(* CoDeSys 2.3.9.48 project: Dev_Test.pro *)
(* Libraries: Standard.lib 20.5.14 08:13:26, Iecsfc.lib 30.1.13 13:05:12, SYSLIBCALLBACK.LIB 30.1.13 13:05:12, WagoLibModbus_IP_01.lib 12.2.16 11:20:24, SysLibSockets.lib 22.5.14 16:16:32, Wago_MBCFG_ETHERNET_01.lib 1.4.15 14:24:28, Wago_MBCFG_COMMON_01.lib 1.4.15 14:24:28 *)

(* PLC configuration (modules and I/O channels)
AT %IX0.0 [BOOLOnX_I] Ch_1 Digital input
AT %IX0.1 [BOOLOnX_I] Ch_2 Digital input
AT %QX4.0 [BOOLOnX_Q] Ch_1 Digital output
AT %QX4.1 [BOOLOnX_Q] Ch_2 Digital output
AT %QW0 [WORDOnW_Q] Ch_1 Analog output
AT %QW1 [WORDOnW_Q] Ch_2 Analog output
AT %QW2 [WORDOnW_Q] Ch_1 Analog output
AT %QW3 [WORDOnW_Q] Ch_2 Analog output
Modbus variables [PFC200MODBUS] node 1, in %IB0 out %QB0 {PlcStopBehaviour = 1; FiledbusErrorBehaviour = 1; TcpOperation = 1; TcpPort = 502; TcpTimeout = 600; UdpOperation = 1; UdpPort = 502; RtuOperation = 0; NodeId = 1; ResponseTimeout = 5000; Interface = 0; Baud = 115200; StopBits = 1; Parity = 1; FlowCtrl = 0; PhysInterface = 0}
Modbus-Master [MB_MASTER] node 2, in %IB0 out %QB0
*)

(* Task configuration *)
TASK NewTask (PRIORITY := 31, INTERVAL := T#1000ms);
	Test();
	SynchronizerModbusStateHandler_PRG();
	SynchroniserSwitch();
	BUS_status_updater();
	MBCFG_ModbusSlave(
	Voltage_LN=> , 
	Power_L=> , 
	MBCFG_IpAddress=> , 
	MBCFG_Port=> , 
	MBCFG_UnitID=> , 
	MBCFG_TimeOut=> , 
	MBCFG_RequestDelay=> , 
	MBCFG_Error=> , 
	MBCFG_LastJob=> );
END_TASK

(* Global variable list: Global_Variables *)
VAR_GLOBAL

	r_modbus_Synchroniser_state								:	REAL:= 1; (* 0 = deny, 1 = allow, 2 = close request*)
	r_modbus_Synchroniser_Denied_Request					:	BOOL;
	r_modbus_Synchroniser_Close_Request					:	BOOL;

	r_DI_Synchroniser_Close_Request				AT %IX0.0	:	BOOL;
	r_DI_Synchroniser_Denied_Request			AT %IX0.1	:	BOOL;

	r_Synchroniser_Close_Request_Relais		AT %QX0.0:	BOOL;
	r_Synchroniser_Close_Denied_Relais			AT %QX0.1:	BOOL; (* only inplemented if hardware output is available *)

(* Offgridbus frequency to analog Out variables*)
     	r_Battery_Bus_Frequency						:	 REAL;
     	x													:	 REAL:=1;
	r_CHP_Power_Control  							: 	REAL;

(* Mixer en CHP frequency variables*)

	Mixer_0_10V_Analog_Control 							AT %QW0		: REAL;
	EV_Charge_0_10V_Analog_Control 					AT %QW1		: REAL;
	CHP_0_20mA_Analog_Control							AT %QW2 		: REAL;


(*Global variables *)
	arSystemState		AT %MW0			:	ARRAY[1.. 2] OF REAL; 			(* Array containing all the system parameters. Values are accessable through modbus tcp starting from register 12288. REAL uses two registers per variable *)



END_VAR

(* POU SWITCHING RELAIS/Test, ST *)
PROGRAM Test
VAR

	Test :fbSwitchRelaysOnOffGrid;
	a: REAL;
	x: REAL;
END_VAR
x := x+1;
arSystemState[1]  := x;

Test(
	r_Off_Grid_Bus_Frequency:= a ,
	r_Off_Grid_Bus_Voltage:= 250,
	r_On_Grid_Start_Frequency:= 49,
	r_On_Grid_Start_Delay_Time:= 2000,
	r_On_Grid_Minimal_On_Time:= 2000 ,
	r_Off_Grid_Start_Frequency:= 51,
	r_Off_Grid_Start_Delay_Time:= 2000,
	r_Switch_Gap_Time:= 2000,
	r_Off_Grid_Minimal_On_Time:= 2000);
END_PROGRAM

(* POU SWITCHING RELAIS/fbSwitchRelaysOnOffGrid, SFC *)
FUNCTION_BLOCK fbSwitchRelaysOnOffGrid
VAR_INPUT

	r_Off_Grid_Bus_Frequency						:	REAL;
	r_Off_Grid_Bus_Voltage							:	REAL;
	r_On_Grid_Start_Frequency						:	REAL;
	r_On_Grid_Start_Delay_Time					:	REAL;
	r_On_Grid_Minimal_On_Time					:	REAL;
	r_Off_Grid_Start_Frequency						:	REAL;
	r_Off_Grid_Start_Delay_Time					:	REAL;
	r_Switch_Gap_Time								: 	REAL;		(* Time between on and off grid relay switching (dead bus gap) *)
	r_Off_Grid_Minimal_On_Time					:	REAL;

END_VAR
VAR_OUTPUT

	r_On_Grid_Relay									:	BOOL;
	r_Off_Grid_Relay									:	BOOL;

END_VAR
VAR

	r_Checked_On_Grid_Start_Frequency			:	REAL;
	r_Checked_Off_Grid_Start_Frequency			:	REAL;

	t_On_Grid_Start_Delay_Timer					:	TON;
	t_Off_Grid_Start_Delay_Timer					:	TON;


END_VAR
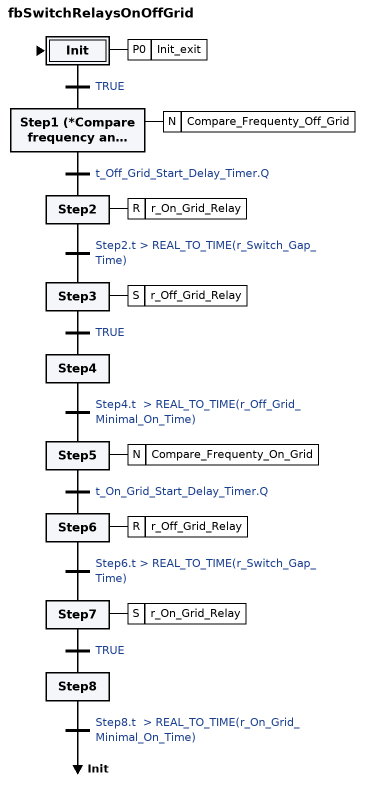
INITIAL_STEP Init:
	Init_exit(P0);
END_STEP
TRANSITION FROM Init TO Step1 (*Compare frequency and voltage *) := TRUE;
END_TRANSITION
STEP Step1 (*Compare frequency and voltage *):
	Compare_Frequenty_Off_Grid(N);
END_STEP
TRANSITION FROM Step1 (*Compare frequency and voltage *) TO Step2 := t_Off_Grid_Start_Delay_Timer.Q;
END_TRANSITION
STEP Step2:
	r_On_Grid_Relay(R);
END_STEP
TRANSITION FROM Step2 TO Step3 := Step2.t > REAL_TO_TIME(r_Switch_Gap_Time);
END_TRANSITION
STEP Step3:
	r_Off_Grid_Relay(S);
END_STEP
TRANSITION FROM Step3 TO Step4 := TRUE;
END_TRANSITION
STEP Step4:
END_STEP
TRANSITION FROM Step4 TO Step5 := Step4.t  > REAL_TO_TIME(r_Off_Grid_Minimal_On_Time);
END_TRANSITION
STEP Step5:
	Compare_Frequenty_On_Grid(N);
END_STEP
TRANSITION FROM Step5 TO Step6 := t_On_Grid_Start_Delay_Timer.Q;
END_TRANSITION
STEP Step6:
	r_Off_Grid_Relay(R);
END_STEP
TRANSITION FROM Step6 TO Step7 := Step6.t > REAL_TO_TIME(r_Switch_Gap_Time);
END_TRANSITION
STEP Step7:
	r_On_Grid_Relay(S);
END_STEP
TRANSITION FROM Step7 TO Step8 := TRUE;
END_TRANSITION
STEP Step8:
END_STEP
TRANSITION FROM Step8 TO Init := Step8.t  > REAL_TO_TIME(r_On_Grid_Minimal_On_Time);
END_TRANSITION

ACTION Init_exit:
(* Off grid frequency should by higher than on grid frequency to prevent pendel behaviour of states *)

IF r_Off_Grid_Start_Frequency > r_On_Grid_Start_Frequency THEN

	r_Checked_Off_Grid_Start_Frequency := r_Off_Grid_Start_Frequency;
	r_Checked_On_Grid_Start_Frequency := r_On_Grid_Start_Frequency;

ELSE

	r_Checked_Off_Grid_Start_Frequency := r_Off_Grid_Start_Frequency;
	r_Checked_On_Grid_Start_Frequency := r_Off_Grid_Start_Frequency;

END_IF
END_ACTION
END_FUNCTION_BLOCK
ACTION Compare_Frequencies:
(* Off grid frequency should by higher than on grid frequency to prevent pendel behaviour of states *)

IF r_Off_Grid_Start_Frequency > r_On_Grid_Start_Frequency THEN

	r_Checked_Off_Grid_Start_Frequency := r_Off_Grid_Start_Frequency;
	r_Checked_On_Grid_Start_Frequency := r_On_Grid_Start_Frequency;

ELSE

	r_Checked_Off_Grid_Start_Frequency := r_Off_Grid_Start_Frequency;
	r_Checked_On_Grid_Start_Frequency := r_Off_Grid_Start_Frequency;

END_IF
END_ACTION
ACTION Compare_Frequenty_Off_Grid:
t_Off_Grid_Start_Delay_Timer(
	IN:= r_Off_Grid_Bus_Frequency > r_Checked_Off_Grid_Start_Frequency AND r_Off_Grid_Bus_Voltage > 150,
	PT:= REAL_TO_TIME(r_On_Grid_Start_Delay_Time));
END_ACTION
ACTION Compare_Frequenty_On_Grid:
t_On_Grid_Start_Delay_Timer(
	IN:= r_Off_Grid_Bus_Frequency < r_Checked_On_Grid_Start_Frequency,
	PT:= REAL_TO_TIME(r_On_Grid_Start_Delay_Time));
END_ACTION

(* POU Switch Synchroniser/SynchronizerModbusStateHandler_PRG, ST *)
PROGRAM SynchronizerModbusStateHandler_PRG
VAR

END_VAR
IF r_modbus_Synchroniser_state < 1 THEN
		r_modbus_Synchroniser_Denied_Request := TRUE;
		r_modbus_Synchroniser_Close_Request := FALSE;
ELSE
	IF r_modbus_Synchroniser_state > 1.99 THEN
		r_modbus_Synchroniser_Denied_Request := FALSE;
		r_modbus_Synchroniser_Close_Request := TRUE;
	ELSE
		r_modbus_Synchroniser_Denied_Request := FALSE;
		r_modbus_Synchroniser_Close_Request := FALSE;
	END_IF
END_IF
END_PROGRAM

(* POU Switch Synchroniser/SynchroniserSwitch, LD *)
PROGRAM SynchroniserSwitch
VAR
END_VAR
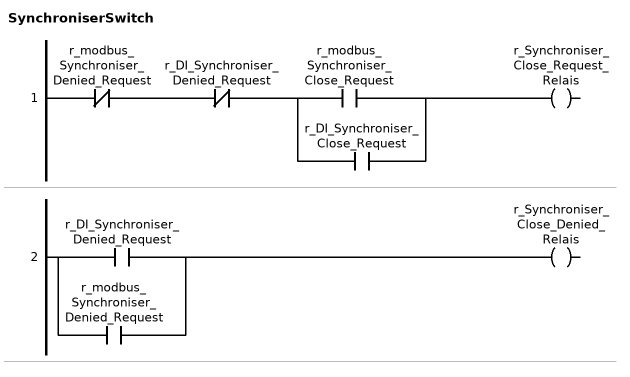
_LD_ (* Ladder Diagram *)
NETWORK 1
	[/r_modbus_Synchroniser_Denied_Request] - [/r_DI_Synchroniser_Denied_Request] - { [r_modbus_Synchroniser_Close_Request] | [r_DI_Synchroniser_Close_Request] } --- (r_Synchroniser_Close_Request_Relais)
NETWORK 2
	{ [r_DI_Synchroniser_Denied_Request] | [r_modbus_Synchroniser_Denied_Request] } --- (r_Synchroniser_Close_Denied_Relais)
_END_LD_
(* the same logic as Structured Text *)
(* Network 1 *)
r_Synchroniser_Close_Request_Relais := NOT r_modbus_Synchroniser_Denied_Request AND NOT r_DI_Synchroniser_Denied_Request AND (r_modbus_Synchroniser_Close_Request OR r_DI_Synchroniser_Close_Request);
(* Network 2 *)
r_Synchroniser_Close_Denied_Relais := r_DI_Synchroniser_Denied_Request OR r_modbus_Synchroniser_Denied_Request;
END_PROGRAM

(* POU Frequency to Analog Out/BUS_status_updater, ST *)
PROGRAM BUS_status_updater
VAR
END_VAR
	(*r_Battery_Bus_Frequency				:=  arMeasurementsGroup1[7];*)
	(* r_Grid_Bus_Frequency					:=  arMeasurementsGroup2[7]; *)

x := x +1;
CHP_Power_Controller();
Mixer_Power_Controller();
EV_Charge_Limit_Controller();
END_PROGRAM

(* POU Frequency to Analog Out/CHP_Power_Controller, FBD *)
PROGRAM CHP_Power_Controller
VAR
	Mixer_to_Frequency_to_Analog_Out: Frequency_to_Analog_Out;
END_VAR
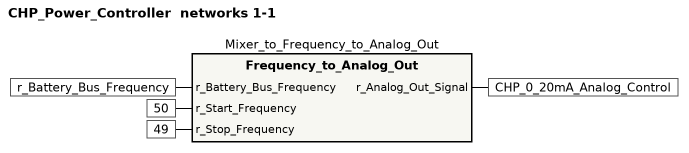
_FBD_ (* Function Block Diagram *)
NETWORK 1 (* Increas the analog output when frequency drops below 50Hz and keeps output at 1 when frequency is below 49Hz *)
	Mixer_to_Frequency_to_Analog_Out:Frequency_to_Analog_Out(r_Battery_Bus_Frequency: r_Battery_Bus_Frequency, r_Start_Frequency: 50, r_Stop_Frequency: 49) => CHP_0_20mA_Analog_Control
_END_FBD_
(* the same logic as Structured Text *)
(* Network 1: Increas the analog output when frequency drops below 50Hz and keeps output at 1 when frequency is below 49Hz *)
Mixer_to_Frequency_to_Analog_Out(r_Battery_Bus_Frequency := r_Battery_Bus_Frequency, r_Start_Frequency := 50, r_Stop_Frequency := 49);
CHP_0_20mA_Analog_Control := Mixer_to_Frequency_to_Analog_Out.r_Analog_Out_Signal;
END_PROGRAM

(* POU Frequency to Analog Out/Frequency_to_Analog_Out, ST *)
FUNCTION_BLOCK Frequency_to_Analog_Out
VAR_INPUT
	r_Battery_Bus_Frequency						:	REAL;
	r_Start_Frequency						:	REAL:=49;
	r_Stop_Frequency						:	REAL:=51;
END_VAR
VAR_OUTPUT
	r_Analog_Out_Signal								:	REAL;
END_VAR
VAR



END_VAR
(* limit control range inbetween start/stop input*)
IF r_Start_Frequency < r_Stop_Frequency THEN
	IF r_Battery_Bus_Frequency < r_Start_Frequency THEN
			r_Battery_Bus_Frequency := r_Start_Frequency;
	END_IF
	IF r_Battery_Bus_Frequency > r_Stop_Frequency THEN
			r_Battery_Bus_Frequency := r_Stop_Frequency;
	END_IF
ELSE
	IF r_Battery_Bus_Frequency > r_Start_Frequency THEN
			r_Battery_Bus_Frequency := r_Start_Frequency;
	END_IF
	IF r_Battery_Bus_Frequency < r_Stop_Frequency THEN
			r_Battery_Bus_Frequency := r_Stop_Frequency;
	END_IF
END_IF

r_Analog_Out_Signal := (r_Battery_Bus_Frequency - r_Start_Frequency) / (r_Stop_Frequency - r_Start_Frequency);
END_FUNCTION_BLOCK

(* POU Frequency to Analog Out/Mixer_Power_Controller, FBD *)
PROGRAM Mixer_Power_Controller
VAR

	CHP_to_Frequency_to_Analog_Out: Frequency_to_Analog_Out;
END_VAR
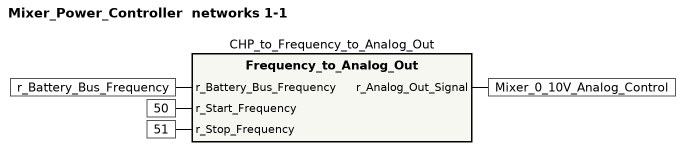
_FBD_ (* Function Block Diagram *)
NETWORK 1
	CHP_to_Frequency_to_Analog_Out:Frequency_to_Analog_Out(r_Battery_Bus_Frequency: r_Battery_Bus_Frequency, r_Start_Frequency: 50, r_Stop_Frequency: 51) => Mixer_0_10V_Analog_Control
_END_FBD_
(* the same logic as Structured Text *)
(* Network 1 *)
CHP_to_Frequency_to_Analog_Out(r_Battery_Bus_Frequency := r_Battery_Bus_Frequency, r_Start_Frequency := 50, r_Stop_Frequency := 51);
Mixer_0_10V_Analog_Control := CHP_to_Frequency_to_Analog_Out.r_Analog_Out_Signal;
END_PROGRAM

(* POU Frequency to Analog Out/EV_Charge_Limit_Controller, FBD *)
PROGRAM EV_Charge_Limit_Controller
VAR

	CHP_to_Frequency_to_Analog_Out: Frequency_to_Analog_Out;
END_VAR
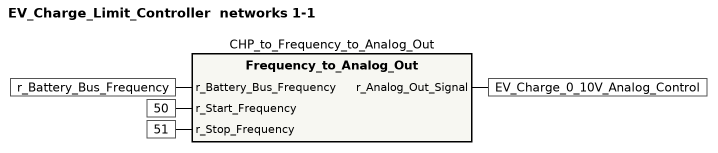
_FBD_ (* Function Block Diagram *)
NETWORK 1
	CHP_to_Frequency_to_Analog_Out:Frequency_to_Analog_Out(r_Battery_Bus_Frequency: r_Battery_Bus_Frequency, r_Start_Frequency: 50, r_Stop_Frequency: 51) => EV_Charge_0_10V_Analog_Control
_END_FBD_
(* the same logic as Structured Text *)
(* Network 1 *)
CHP_to_Frequency_to_Analog_Out(r_Battery_Bus_Frequency := r_Battery_Bus_Frequency, r_Start_Frequency := 50, r_Stop_Frequency := 51);
EV_Charge_0_10V_Analog_Control := CHP_to_Frequency_to_Analog_Out.r_Analog_Out_Signal;
END_PROGRAM

(* POU Generated Code/Ethernet/MBCFG_ModbusSlave, ST *)
PROGRAM MBCFG_ModbusSlave(* generated by config one prg for each slave *)

VAR_INPUT

END_VAR

VAR_OUTPUT
       Voltage_LN       :    REAL;       (*Voltage L-N  _G_ULN[0]*) 
       Power_L       :    REAL;       (*Real Power L   _G_PLN[0]*) 

    (*--- system variables (read only) ----------------------------------------*)
    MBCFG_IpAddress     :   STRING(7) := '0.0.0.0'; (* address of this slave *)
    MBCFG_Port          :   UINT := 502;               (* IP - Port *)
    MBCFG_UnitID        :   BYTE := 0;             (* MODBUS Unit-Id *)
    MBCFG_TimeOut       :   TIME := t#20ms;           (* Response timeout*)
	MBCFG_RequestDelay  :   TIME  := t#0ms;         (* 0 means no delay *)
    MBCFG_Error         :   MBCFG_eERROR := MBCFG_START_UP;
	MBCFG_LastJob       :   MBCFG_typCOM_JOB;
    (*-------------------------------------------------------------------------*)
END_VAR

{library private}
VAR CONSTANT
    zz_VARIABLECOUNT:   INT := 2; (* number of variables  *)
    zz_JOBCOUNT     :   INT := 2; (* number of jobs *)
END_VAR
VAR

    (*=== VARIABLE LIST ===============================================================================*)
    zz_VariableList :   ARRAY[1..zz_VARIABLECOUNT] OF MBCFG_typVARIABLE :=
    (    DataType        := MBCFG_TYPE_REAL,
        ByteOrder       := MBCFG_BYTE_ORDER_0,
        BitSize         := 32,
        ptVar           := 0,
        ReadJobIndex    := 1,
        ReadStartBitNo  := 0,
        WriteJobIndex   := 0,
        WriteStartBitNo := 0 ),
    (    DataType        := MBCFG_TYPE_REAL,
        ByteOrder       := MBCFG_BYTE_ORDER_0,
        BitSize         := 32,
        ptVar           := 0,
        ReadJobIndex    := 2,
        ReadStartBitNo  := 0,
        WriteJobIndex   := 0,
        WriteStartBitNo := 0 )

                        ;
    (*=================================================================================================*)

    (*=== JOB LIST ====================================================================================*)
    zz_JobList     :   ARRAY[1..zz_JOBCOUNT] OF MBCFG_typCOM_JOB :=
     (   Functioncode            := 3,
        ReadStartAddress        := 19000,
        ReadQuantity            := 2,
        WriteStartAddress       := 0,
        WriteQuantity           := 0,
        ptReadData              := 0, 
        ptWriteData             := 0 ),
     (   Functioncode            := 3,
        ReadStartAddress        := 19020,
        ReadQuantity            := 2,
        WriteStartAddress       := 0,
        WriteQuantity           := 0,
        ptReadData              := 0, 
        ptWriteData             := 0 )

                        ;
    (*=================================================================================================*)

    (*=== DATA FIELDS =================================================================================*)
     zz_DataField_1_Read       :       ARRAY[1..2] OF WORD;
     zz_DataField_2_Read       :       ARRAY[1..2] OF WORD;
	
    (*=================================================================================================*)

    (*=== MODBUS MASTER =====================================*)
    zz_MBCFG_MASTER_ETH :       MBCFG_MASTER_TCP;
    (*=======================================================*)

END_VAR
(*--- for each variable -------------------------*)
   zz_VariableList[1].ptVar := ADR(Voltage_LN);
   zz_VariableList[2].ptVar := ADR(Power_L);

(*-----------------------------------------------*)

(*--- for each job -----------------------------------*)
zz_JobList[1].ptReadData   := ADR(zz_DataField_1_Read);
zz_JobList[2].ptReadData   := ADR(zz_DataField_2_Read);

(*----------------------------------------------------*)


(*#### START OF FIXED CODE #####################################*)
zz_MBCFG_MASTER_ETH(	strIpAddress    := MBCFG_IpAddress,                 (* fixed entry     *)
                        uiPort          := MBCFG_Port,                      (* fixed entry     *)
                        bUnitID         := MBCFG_UnitID,                    (* fixed entry     *)
                        tTimeOut        := MBCFG_TimeOut,                   (* fixed entry     *)
                        iVariableCount  := zz_VARIABLECOUNT,
                        ptVariableList  := ADR(zz_VariableList),
                        iJobCount       := zz_JOBCOUNT,
                        ptJobList       := ADR(zz_JobList),
                        tRequestDelay   := MBCFG_RequestDelay,              (* fixed entry     *)
                        eError          => MBCFG_Error,                     (* fixed entry     *)
                        LastJob         => MBCFG_LastJob                    (* fixed entry     *)
                    );
(*##############################################################*)
END_PROGRAM

(* POU Configuration/MODBUS_CONFIGURATION, ST *)
PROGRAM MODBUS_CONFIGURATION
VAR                                
END_VAR                            
(*
   <?xml version="1.0" encoding="UTF-16" standalone="yes"?>
<network xml_structure_version="1" xml_feature_version="1">
	<generator_settings minRTUTaskCycleTimeMs="5" minEthaskCycleTimeMs="5" ethSlaveMultiplier="0.1" rtuInterfaceMultiplier="0.1" taskGeneration="false"/>
	<master_interface type="eth" name="" expanded="true">
		<mb_slave comment="" name="ModbusSlave" expanded="true" type="generic">
			<mb_connection type="eth" transport="TCP" port="502" ip="0.0.0.0" unitid="0" request_delay_ms="0" response_timeout_ms="20"/>
			<generic_vars comment="" expanded="true">
				<generic_var data_type="REAL">
					<generic_params name="Voltage_LN" comment="Voltage L-N  _G_ULN[0]" expanded="false" mb_iotype="unused" mb_access="ro" var_byteorder="B1B2B3B4"/>
					<mb_address explicitAccess="false" FCRead="3" FCWrite="0" ReadMBAddress="19000" WriteMBAddress="0" ReadBitOffset="0" WriteBitOffset="0"/>
				</generic_var>
				<generic_var data_type="REAL">
					<generic_params name="Power_L" comment="Real Power L   _G_PLN[0]" expanded="true" mb_iotype="unused" mb_access="ro" var_byteorder="B1B2B3B4"/>
					<mb_address explicitAccess="false" FCRead="3" FCWrite="0" ReadMBAddress="19020" WriteMBAddress="0" ReadBitOffset="0" WriteBitOffset="0"/>
				</generic_var>
			</generic_vars>
		</mb_slave>
	</master_interface>
</network>
                              
*)                                 
;                                  
END_PROGRAM
